{attribute 'GeneratedUsingTerminal: EL7332-0000-0024'}
{attribute addProperty BoxType "EL7332-0000-0024"}
{attribute addProperty Id "EnableBOOL1ResetBOOL1Reduce_torqueBOOL1"}
{attribute addProperty CRC "3376996594"}
{attribute addProperty Size "3"}
TYPE Control_C948E0F2 :
STRUCT
    {attribute addProperty Name "Enable"}
    Enable : BOOL;
    {attribute addProperty Name "Reset"}
    Reset : BOOL;
    {attribute addProperty Name "Reduce_torque"}
    Reduce_torque : BOOL;
END_STRUCT
END_TYPE

(* stored: Version 1.2.0.0, ProductVersion 3.1.4024.11
   DUT Control_C948E0F2: Id {4c1b433c-61bf-0bad-3aa4-0f80ec0144ca} *)
